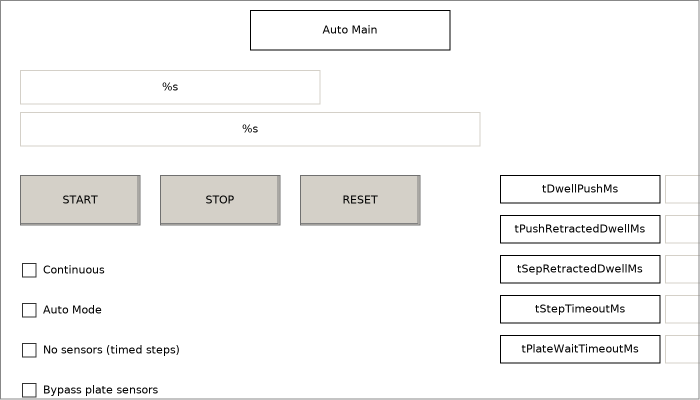
VISUALIZATION AutoMain  // 700x400
VAR_IN_OUT
	stMasterAutoCycle : ST_HmiMasterAuto;
	stCfg : ST_HmiMasterAutoCfg;
END_VAR
    Rectangle (250,10 200x40), "Auto Main"
    Textfield (20,70 300x34), "%s", text variable: stMasterAutoCycle.sStepText
    Textfield (20,112 460x34), "%s", text variable: stMasterAutoCycle.sErrorText
    Button (20,175 120x50), "START"
        tap stMasterAutoCycle.bStart
    Button (160,175 120x50), "STOP"
        tap stMasterAutoCycle.bStop
    Button (300,175 120x50), "RESET"
        tap stMasterAutoCycle.bReset
    Checkbox (20,255 240x30), "Continuous", variable: stCfg.bContinuous
    Checkbox (20,295 240x30), "Auto Mode", variable: stCfg.bAutoMode
    Checkbox (20,335 240x30), "No sensors (timed steps)", variable: stCfg.bNoSensors
    Checkbox (20,375 240x30), "Bypass plate sensors", variable: stCfg.bBypassPlateSensors
    Rectangle (500,175 160x28), "tDwellPushMs"
    Textfield (665,175 115x28), "%d", text variable: stCfg.tDwellPushMs
        OnMouseClick: write the text variable via Default
    Rectangle (500,215 160x28), "tPushRetractedDwellMs"
    Textfield (665,215 115x28), "%d", text variable: stCfg.tPushRetractedDwellMs
        OnMouseClick: write the text variable via Default
    Rectangle (500,255 160x28), "tSepRetractedDwellMs"
    Textfield (665,255 115x28), "%d", text variable: stCfg.tSepRetractedDwellMs
        OnMouseClick: write the text variable via Default
    Rectangle (500,295 160x28), "tStepTimeoutMs"
    Textfield (665,295 115x28), "%d", text variable: stCfg.tStepTimeoutMs
        OnMouseClick: write the text variable via Default
    Rectangle (500,335 160x28), "tPlateWaitTimeoutMs"
    Textfield (665,335 115x28), "%d", text variable: stCfg.tPlateWaitTimeoutMs
        OnMouseClick: write the text variable via Default
END_VISUALIZATION

(* stored: Version 1.1.0.1, ProductVersion 3.1.4024.16
   Visu AutoMain: Id {5cb01f7a-eb2a-41a3-a05b-192e39796768} *)
